PROGRAM Powerall
VAR
	Powerall : FB_PowerAll;
END_VAR

Powerall(enable := True);

END_PROGRAM

(* stored: Version 1.1.0.1, ProductVersion 3.1.0.25
   POU Powerall: Id {9293db3e-56c7-463a-b7a8-0f329de9d653} *)
